FUNCTION_BLOCK AnlagenSequenz_06 (* Ring aus getrennter Vorlauf- und Nachlauf-Kette (je 5 Zwischenschritte) für 6 Motoren mit Störungs-Kaskade, s. KONZEPT_Anlagensequenz.md *)
  (* Standard: 61499-2; ApplicationDomain: Fördertechnik; Description: Copyright (c) 2026 HR Agrartechnik GmbH This program and the accompanying materials are made available under the terms of the Eclipse Public License 2.0 which is available at https://www.eclipse.org/legal/epl-2.0/ SPDX-License-Identifier: EPL-2.0 DRAFT (2026-08-12), 2. Fassung: Vorlauf und Nachlauf sind jetzt zwei getrennte, jeweils rein lineare Ketten (S_VOR1..S_VOR5 bzw. S_NACH1..S_NACH5), verbunden über S_AUS (unten) und S_LAEUFT (oben) zu einem Ring - anstelle der ersten Fassung mit 7 bidirektional genutzten Zuständen. Jeder Zustand hat dadurch genau einen festen Zeitwert (ZEk_EIN bzw. ZEk_AUS) und ein festes Motor-Muster, keine Richtungs-Fallunterscheidung mehr pro Zustand nötig. Bekannte, bewusste Vereinfachungen: 1) Jede STOERUNG_Mx hat ein eigenes Event EI_Mx (analog EO_Mx/DO_Mx), das direkt von jedem Zustand vor dem jeweiligen Zielschritt (S_NACH_x, bzw. S_AUS bei x=6) dorthin springt - kein Umweg mehr über einen Spiegelpunkt und kein Nachfassen über mehrere Zyklen. Ein AUS-Abbruch aus dem Vorlauf springt weiterhin auf den Spiegelpunkt (S_VOR_k -> S_NACH_(6-k)), da dort keine Motoren-Störung, sondern nur der Bedienerwunsch vorliegt. 2) Pro Motor gibt es ein Event EO_Mx mit angehängtem DO_Mx (analog EO_Sx/DO_Sx in sequence_T_04/_08). Der Baustein hat keine Selbstschleifen mehr (alle bisherigen liefen über das inzwischen entfernte EI_CYCLIC) - EO_Mx feuert also nur noch bei einem echten Zustandswechsel. 3) MaxBetriebRest/Nachlauf-Reste (Demo-Server-Schema) sind noch nicht abgebildet. *)
  (* Version 0.6, 2026-08-12, Franz Höpfinger, HR Agrartechnik GmbH *)
  PACKAGE logiBUS::utils::sequence::timed;
  IMPORT logiBUS::utils::sequence::const::sequence;
  IMPORT logiBUS::utils::sequence::const::sequence::NO_TIME;
  IMPORT logiBUS::utils::sequence::const::anlagenSequenz;
  IMPORT logiBUS::utils::sequence::const::anlagenSequenz::STATUS_BETRIEB_AUS;
  IMPORT logiBUS::utils::sequence::const::anlagenSequenz::STATUS_BETRIEB_HOCHFAHREN;
  IMPORT logiBUS::utils::sequence::const::anlagenSequenz::STATUS_BETRIEB_LAEUFT;
  IMPORT logiBUS::utils::sequence::const::anlagenSequenz::STATUS_BETRIEB_HERUNTERFAHREN;
  IMPORT logiBUS::utils::sequence::const::anlagenSequenz::STATUS_STOERUNG_KEINE;
  IMPORT logiBUS::utils::sequence::const::anlagenSequenz::STATUS_STOERUNG_AKTIV;
  IMPORT logiBUS::utils::sequence::const::anlagenSequenz::TRANSIT_ART_KEINE;
  IMPORT logiBUS::utils::sequence::const::anlagenSequenz::TRANSIT_ART_VORLAUF;
  IMPORT logiBUS::utils::sequence::const::anlagenSequenz::TRANSIT_ART_NACHLAUF;
  IMPORT logiBUS::utils::sequence::const::motorNummer;
  IMPORT logiBUS::utils::sequence::const::motorNummer::MOTOR_KEINER;
  IMPORT logiBUS::utils::sequence::const::motorNummer::MOTOR_M1;
  IMPORT logiBUS::utils::sequence::const::motorNummer::MOTOR_M2;
  IMPORT logiBUS::utils::sequence::const::motorNummer::MOTOR_M3;
  IMPORT logiBUS::utils::sequence::const::motorNummer::MOTOR_M4;
  IMPORT logiBUS::utils::sequence::const::motorNummer::MOTOR_M5;
  IMPORT logiBUS::utils::sequence::const::motorNummer::MOTOR_M6;
  IMPORT logiBUS::utils::sequence::const::zaehlstand;
  IMPORT logiBUS::utils::sequence::const::zaehlstand::ZAEHLSTAND_0;
  IMPORT logiBUS::utils::sequence::const::zaehlstand::ZAEHLSTAND_1;
  IMPORT logiBUS::utils::sequence::const::zaehlstand::ZAEHLSTAND_2;
  IMPORT logiBUS::utils::sequence::const::zaehlstand::ZAEHLSTAND_3;
  IMPORT logiBUS::utils::sequence::const::zaehlstand::ZAEHLSTAND_4;
  IMPORT logiBUS::utils::sequence::const::zaehlstand::ZAEHLSTAND_5;
  IMPORT logiBUS::utils::sequence::const::zaehlstand::ZAEHLSTAND_6;
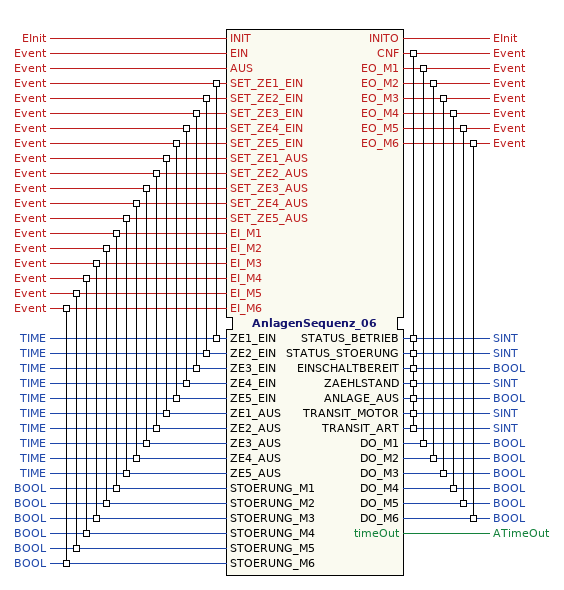
  EVENT_INPUT
    INIT : EInit; (* Initialization Request *)
    EIN; (* Startsequenz auslösen; nur wirksam wenn EINSCHALTBEREIT=TRUE; quittiert dabei zugleich eine anstehende Störungsanzeige *)
    AUS; (* Stopsequenz auslösen, aus jedem Schritt der Vorlauf-Kette oder aus S_LAEUFT *)
    SET_ZE1_EIN WITH ZE1_EIN; (* Update ZE1_EIN independently of EIN *)
    SET_ZE2_EIN WITH ZE2_EIN; (* Update ZE2_EIN independently of EIN *)
    SET_ZE3_EIN WITH ZE3_EIN; (* Update ZE3_EIN independently of EIN *)
    SET_ZE4_EIN WITH ZE4_EIN; (* Update ZE4_EIN independently of EIN *)
    SET_ZE5_EIN WITH ZE5_EIN; (* Update ZE5_EIN independently of EIN *)
    SET_ZE1_AUS WITH ZE1_AUS; (* Update ZE1_AUS independently of AUS *)
    SET_ZE2_AUS WITH ZE2_AUS; (* Update ZE2_AUS independently of AUS *)
    SET_ZE3_AUS WITH ZE3_AUS; (* Update ZE3_AUS independently of AUS *)
    SET_ZE4_AUS WITH ZE4_AUS; (* Update ZE4_AUS independently of AUS *)
    SET_ZE5_AUS WITH ZE5_AUS; (* Update ZE5_AUS independently of AUS *)
    EI_M1 WITH STOERUNG_M1; (* Störungsstatus Motor 1 hat sich geändert *)
    EI_M2 WITH STOERUNG_M2; (* Störungsstatus Motor 2 hat sich geändert *)
    EI_M3 WITH STOERUNG_M3; (* Störungsstatus Motor 3 hat sich geändert *)
    EI_M4 WITH STOERUNG_M4; (* Störungsstatus Motor 4 hat sich geändert *)
    EI_M5 WITH STOERUNG_M5; (* Störungsstatus Motor 5 hat sich geändert *)
    EI_M6 WITH STOERUNG_M6; (* Störungsstatus Motor 6 hat sich geändert *)
  END_EVENT
  EVENT_OUTPUT
    INITO : EInit; (* Initialization Confirm *)
    CNF WITH STATUS_BETRIEB, STATUS_STOERUNG, ZAEHLSTAND, EINSCHALTBEREIT, ANLAGE_AUS, TRANSIT_MOTOR, TRANSIT_ART; (* Ausführungsbestätigung, mit jedem Zustands-Update *)
    EO_M1 WITH DO_M1; (* Laufbefehl Motor 1 aktualisiert (analog EO_Sx in sequence_T_04/_08) *)
    EO_M2 WITH DO_M2; (* Laufbefehl Motor 2 aktualisiert *)
    EO_M3 WITH DO_M3; (* Laufbefehl Motor 3 aktualisiert *)
    EO_M4 WITH DO_M4; (* Laufbefehl Motor 4 aktualisiert *)
    EO_M5 WITH DO_M5; (* Laufbefehl Motor 5 aktualisiert *)
    EO_M6 WITH DO_M6; (* Laufbefehl Motor 6 aktualisiert *)
  END_EVENT
  VAR_INPUT
    ZE1_EIN : TIME := sequence::NO_TIME; (* S_VOR1 zu S_VOR2, M5 startet (Vorlauf) *)
    ZE2_EIN : TIME := sequence::NO_TIME; (* S_VOR2 zu S_VOR3, M4 startet (Vorlauf) *)
    ZE3_EIN : TIME := sequence::NO_TIME; (* S_VOR3 zu S_VOR4, M3 startet (Vorlauf) *)
    ZE4_EIN : TIME := sequence::NO_TIME; (* S_VOR4 zu S_VOR5, M2 startet (Vorlauf) *)
    ZE5_EIN : TIME := sequence::NO_TIME; (* S_VOR5 zu S_LAEUFT, M1 startet (Vorlauf) *)
    ZE1_AUS : TIME := sequence::NO_TIME; (* S_NACH1 zu S_NACH2, M2 stoppt (Nachlauf) *)
    ZE2_AUS : TIME := sequence::NO_TIME; (* S_NACH2 zu S_NACH3, M3 stoppt (Nachlauf) *)
    ZE3_AUS : TIME := sequence::NO_TIME; (* S_NACH3 zu S_NACH4, M4 stoppt (Nachlauf) *)
    ZE4_AUS : TIME := sequence::NO_TIME; (* S_NACH4 zu S_NACH5, M5 stoppt (Nachlauf) *)
    ZE5_AUS : TIME := sequence::NO_TIME; (* S_NACH5 zu S_AUS, M6 stoppt (Nachlauf) *)
    STOERUNG_M1 : BOOL := BOOL#FALSE; (* Motor 1 hat aktuell eine Störung anstehen *)
    STOERUNG_M2 : BOOL := BOOL#FALSE; (* Motor 2 hat aktuell eine Störung anstehen *)
    STOERUNG_M3 : BOOL := BOOL#FALSE; (* Motor 3 hat aktuell eine Störung anstehen *)
    STOERUNG_M4 : BOOL := BOOL#FALSE; (* Motor 4 hat aktuell eine Störung anstehen *)
    STOERUNG_M5 : BOOL := BOOL#FALSE; (* Motor 5 hat aktuell eine Störung anstehen *)
    STOERUNG_M6 : BOOL := BOOL#FALSE; (* Motor 6 hat aktuell eine Störung anstehen *)
  END_VAR
  VAR_OUTPUT
    STATUS_BETRIEB : SINT; (* 0=Aus 1=Hochfahren 2=Läuft 3=Herunterfahren *)
    STATUS_STOERUNG : SINT; (* 0=keine 4=aktiv, verriegelt bis EIN *)
    EINSCHALTBEREIT : BOOL; (* TRUE nur wenn alle Motoren stehen UND alle Motoren störungsfrei sind *)
    ZAEHLSTAND : SINT; (* 0..6, Anzahl aktuell laufender Motoren, s. Konzept *)
    ANLAGE_AUS : BOOL; (* TRUE nur in S_AUS (STATUS_BETRIEB = Aus) - Voraussetzung fuer Handbetrieb *)
    TRANSIT_MOTOR : SINT; (* 0 = keiner (S_AUS/S_LAEUFT), 1..6 = Motor-Nr., der nach Ablauf der aktuellen Zeit startet/stoppt (siehe TRANSIT_ART) *)
    TRANSIT_ART : SINT; (* anlagenSequenz::TRANSIT_ART_KEINE/_VORLAUF/_NACHLAUF *)
    DO_M1 : BOOL; (* Laufbefehl Motor 1 *)
    DO_M2 : BOOL; (* Laufbefehl Motor 2 *)
    DO_M3 : BOOL; (* Laufbefehl Motor 3 *)
    DO_M4 : BOOL; (* Laufbefehl Motor 4 *)
    DO_M5 : BOOL; (* Laufbefehl Motor 5 *)
    DO_M6 : BOOL; (* Laufbefehl Motor 6 *)
  END_VAR
  PLUGS
    timeOut : iec61499::events::ATimeOut; (* timeOut Adapter *)
  END_PLUGS
  EC_STATES
    xSTART; (* Initial State *)
    Init : -> INITO; (* Initialization *)
    sAUS : S_AUS_Setup, EI_CYCLIC_Auswertung, M1_AUS -> EO_M1, M2_AUS -> EO_M2, M3_AUS -> EO_M3, M4_AUS -> EO_M4, M5_AUS -> EO_M5, M6_AUS -> EO_M6, -> CNF; (* S_AUS, unten im Ring: keine Motoren laufen *)
    sVOR1 : S_VOR1_Setup, EI_CYCLIC_Auswertung, M1_AUS -> EO_M1, M2_AUS -> EO_M2, M3_AUS -> EO_M3, M4_AUS -> EO_M4, M5_AUS -> EO_M5, M6_EIN -> EO_M6, -> timeOut.START, -> CNF; (* S_VOR1 (Vorlauf-Kette): nur M6 läuft *)
    sVOR2 : S_VOR2_Setup, EI_CYCLIC_Auswertung, M1_AUS -> EO_M1, M2_AUS -> EO_M2, M3_AUS -> EO_M3, M4_AUS -> EO_M4, M5_EIN -> EO_M5, M6_EIN -> EO_M6, -> timeOut.START, -> CNF; (* S_VOR2 (Vorlauf-Kette): M5,M6 laufen *)
    sVOR3 : S_VOR3_Setup, EI_CYCLIC_Auswertung, M1_AUS -> EO_M1, M2_AUS -> EO_M2, M3_AUS -> EO_M3, M4_EIN -> EO_M4, M5_EIN -> EO_M5, M6_EIN -> EO_M6, -> timeOut.START, -> CNF; (* S_VOR3 (Vorlauf-Kette): M4,M5,M6 laufen *)
    sVOR4 : S_VOR4_Setup, EI_CYCLIC_Auswertung, M1_AUS -> EO_M1, M2_AUS -> EO_M2, M3_EIN -> EO_M3, M4_EIN -> EO_M4, M5_EIN -> EO_M5, M6_EIN -> EO_M6, -> timeOut.START, -> CNF; (* S_VOR4 (Vorlauf-Kette): M3,M4,M5,M6 laufen *)
    sVOR5 : S_VOR5_Setup, EI_CYCLIC_Auswertung, M1_AUS -> EO_M1, M2_EIN -> EO_M2, M3_EIN -> EO_M3, M4_EIN -> EO_M4, M5_EIN -> EO_M5, M6_EIN -> EO_M6, -> timeOut.START, -> CNF; (* S_VOR5 (Vorlauf-Kette): M2,M3,M4,M5,M6 laufen *)
    sLAEUFT : S_LAEUFT_Setup, EI_CYCLIC_Auswertung, M1_EIN -> EO_M1, M2_EIN -> EO_M2, M3_EIN -> EO_M3, M4_EIN -> EO_M4, M5_EIN -> EO_M5, M6_EIN -> EO_M6, -> CNF; (* S_LAEUFT, oben im Ring: alle 6 Motoren laufen *)
    sNACH1 : S_NACH1_Setup, EI_CYCLIC_Auswertung, M1_AUS -> EO_M1, M2_EIN -> EO_M2, M3_EIN -> EO_M3, M4_EIN -> EO_M4, M5_EIN -> EO_M5, M6_EIN -> EO_M6, -> timeOut.START, -> CNF; (* S_NACH1 (Nachlauf-Kette): M2,M3,M4,M5,M6 laufen (M1 gestoppt) *)
    sNACH2 : S_NACH2_Setup, EI_CYCLIC_Auswertung, M1_AUS -> EO_M1, M2_AUS -> EO_M2, M3_EIN -> EO_M3, M4_EIN -> EO_M4, M5_EIN -> EO_M5, M6_EIN -> EO_M6, -> timeOut.START, -> CNF; (* S_NACH2 (Nachlauf-Kette): M3,M4,M5,M6 laufen *)
    sNACH3 : S_NACH3_Setup, EI_CYCLIC_Auswertung, M1_AUS -> EO_M1, M2_AUS -> EO_M2, M3_AUS -> EO_M3, M4_EIN -> EO_M4, M5_EIN -> EO_M5, M6_EIN -> EO_M6, -> timeOut.START, -> CNF; (* S_NACH3 (Nachlauf-Kette): M4,M5,M6 laufen *)
    sNACH4 : S_NACH4_Setup, EI_CYCLIC_Auswertung, M1_AUS -> EO_M1, M2_AUS -> EO_M2, M3_AUS -> EO_M3, M4_AUS -> EO_M4, M5_EIN -> EO_M5, M6_EIN -> EO_M6, -> timeOut.START, -> CNF; (* S_NACH4 (Nachlauf-Kette): M5,M6 laufen *)
    sNACH5 : S_NACH5_Setup, EI_CYCLIC_Auswertung, M1_AUS -> EO_M1, M2_AUS -> EO_M2, M3_AUS -> EO_M3, M4_AUS -> EO_M4, M5_AUS -> EO_M5, M6_EIN -> EO_M6, -> timeOut.START, -> CNF; (* S_NACH5 (Nachlauf-Kette): nur M6 läuft *)
  END_STATES
  EC_TRANSITIONS
    sAUS TO sVOR1 := EIN[NOT (STOERUNG_M1 OR STOERUNG_M2 OR STOERUNG_M3 OR STOERUNG_M4 OR STOERUNG_M5 OR STOERUNG_M6)];
    sVOR1 TO sVOR2 := timeOut.TimeOut;
    sVOR1 TO sNACH5 := AUS;
    sVOR1 TO sNACH1 := EI_M1[STOERUNG_M1];
    sVOR1 TO sNACH2 := EI_M2[STOERUNG_M2];
    sVOR1 TO sNACH3 := EI_M3[STOERUNG_M3];
    sVOR1 TO sNACH4 := EI_M4[STOERUNG_M4];
    sVOR1 TO sNACH5 := EI_M5[STOERUNG_M5];
    sVOR1 TO sAUS := EI_M6[STOERUNG_M6];
    sVOR2 TO sVOR3 := timeOut.TimeOut;
    sVOR2 TO sNACH4 := AUS;
    sVOR2 TO sNACH1 := EI_M1[STOERUNG_M1];
    sVOR2 TO sNACH2 := EI_M2[STOERUNG_M2];
    sVOR2 TO sNACH3 := EI_M3[STOERUNG_M3];
    sVOR2 TO sNACH4 := EI_M4[STOERUNG_M4];
    sVOR2 TO sNACH5 := EI_M5[STOERUNG_M5];
    sVOR2 TO sAUS := EI_M6[STOERUNG_M6];
    sVOR3 TO sVOR4 := timeOut.TimeOut;
    sVOR3 TO sNACH3 := AUS;
    sVOR3 TO sNACH1 := EI_M1[STOERUNG_M1];
    sVOR3 TO sNACH2 := EI_M2[STOERUNG_M2];
    sVOR3 TO sNACH3 := EI_M3[STOERUNG_M3];
    sVOR3 TO sNACH4 := EI_M4[STOERUNG_M4];
    sVOR3 TO sNACH5 := EI_M5[STOERUNG_M5];
    sVOR3 TO sAUS := EI_M6[STOERUNG_M6];
    sVOR4 TO sVOR5 := timeOut.TimeOut;
    sVOR4 TO sNACH2 := AUS;
    sVOR4 TO sNACH1 := EI_M1[STOERUNG_M1];
    sVOR4 TO sNACH2 := EI_M2[STOERUNG_M2];
    sVOR4 TO sNACH3 := EI_M3[STOERUNG_M3];
    sVOR4 TO sNACH4 := EI_M4[STOERUNG_M4];
    sVOR4 TO sNACH5 := EI_M5[STOERUNG_M5];
    sVOR4 TO sAUS := EI_M6[STOERUNG_M6];
    sVOR5 TO sLAEUFT := timeOut.TimeOut;
    sVOR5 TO sNACH1 := AUS;
    sVOR5 TO sNACH1 := EI_M1[STOERUNG_M1];
    sVOR5 TO sNACH2 := EI_M2[STOERUNG_M2];
    sVOR5 TO sNACH3 := EI_M3[STOERUNG_M3];
    sVOR5 TO sNACH4 := EI_M4[STOERUNG_M4];
    sVOR5 TO sNACH5 := EI_M5[STOERUNG_M5];
    sVOR5 TO sAUS := EI_M6[STOERUNG_M6];
    sLAEUFT TO sNACH1 := AUS;
    sLAEUFT TO sNACH1 := EI_M1[STOERUNG_M1];
    sLAEUFT TO sNACH2 := EI_M2[STOERUNG_M2];
    sLAEUFT TO sNACH3 := EI_M3[STOERUNG_M3];
    sLAEUFT TO sNACH4 := EI_M4[STOERUNG_M4];
    sLAEUFT TO sNACH5 := EI_M5[STOERUNG_M5];
    sLAEUFT TO sAUS := EI_M6[STOERUNG_M6];
    sNACH1 TO sNACH2 := timeOut.TimeOut;
    sNACH1 TO sNACH2 := EI_M2[STOERUNG_M2];
    sNACH1 TO sNACH3 := EI_M3[STOERUNG_M3];
    sNACH1 TO sNACH4 := EI_M4[STOERUNG_M4];
    sNACH1 TO sNACH5 := EI_M5[STOERUNG_M5];
    sNACH1 TO sAUS := EI_M6[STOERUNG_M6];
    sNACH2 TO sNACH3 := timeOut.TimeOut;
    sNACH2 TO sNACH3 := EI_M3[STOERUNG_M3];
    sNACH2 TO sNACH4 := EI_M4[STOERUNG_M4];
    sNACH2 TO sNACH5 := EI_M5[STOERUNG_M5];
    sNACH2 TO sAUS := EI_M6[STOERUNG_M6];
    sNACH3 TO sNACH4 := timeOut.TimeOut;
    sNACH3 TO sNACH4 := EI_M4[STOERUNG_M4];
    sNACH3 TO sNACH5 := EI_M5[STOERUNG_M5];
    sNACH3 TO sAUS := EI_M6[STOERUNG_M6];
    sNACH4 TO sNACH5 := timeOut.TimeOut;
    sNACH4 TO sNACH5 := EI_M5[STOERUNG_M5];
    sNACH4 TO sAUS := EI_M6[STOERUNG_M6];
    sNACH5 TO sAUS := timeOut.TimeOut;
    sNACH5 TO sAUS := EI_M6[STOERUNG_M6];
    sVOR1 TO sVOR1 := SET_ZE1_EIN;
    sVOR2 TO sVOR2 := SET_ZE2_EIN;
    sVOR3 TO sVOR3 := SET_ZE3_EIN;
    sVOR4 TO sVOR4 := SET_ZE4_EIN;
    sVOR5 TO sVOR5 := SET_ZE5_EIN;
    sNACH1 TO sNACH1 := SET_ZE1_AUS;
    sNACH2 TO sNACH2 := SET_ZE2_AUS;
    sNACH3 TO sNACH3 := SET_ZE3_AUS;
    sNACH4 TO sNACH4 := SET_ZE4_AUS;
    sNACH5 TO sNACH5 := SET_ZE5_AUS;
    xSTART TO Init := INIT;
    Init TO sAUS := 1;
  END_TRANSITIONS
  ALGORITHM initialize IN ST: (* Initialization algorithm *)

  END_ALGORITHM
  ALGORITHM deInitialize IN ST: (* Normally executed algorithm *)

  END_ALGORITHM
  ALGORITHM EI_CYCLIC_Auswertung IN ST: (* Liest STOERUNG_M1..M6 neu ein, setzt STATUS_STOERUNG falls eine aktiv ist, und berechnet EINSCHALTBEREIT/ANLAGE_AUS *)
// Störungssignale frisch einlesen (BOOL-Dauersignale, kein Event-Consumption-Problem, s. Konzept
// Frage 4)
IF STOERUNG_M1 OR STOERUNG_M2 OR STOERUNG_M3 OR STOERUNG_M4 OR STOERUNG_M5 OR STOERUNG_M6 THEN
	STATUS_STOERUNG := anlagenSequenz::STATUS_STOERUNG_AKTIV; // verriegelt bis zur nächsten erfolgreichen EIN-Quittierung
END_IF;

// Einschaltbereit: alle Motoren stehen (S_AUS) UND alle Motoren aktuell (live) störungsfrei.
// Bewusst NICHT an STATUS_STOERUNG gekoppelt: das bleibt bis zum naechsten EIN verriegelt, EIN
// selbst kommt aber nur an, wenn EINSCHALTBEREIT die Visu-Sperre freigibt - sonst Deadlock.
EINSCHALTBEREIT := (ZAEHLSTAND = 0)
	AND NOT (STOERUNG_M1 OR STOERUNG_M2 OR STOERUNG_M3 OR STOERUNG_M4 OR STOERUNG_M5 OR STOERUNG_M6);

// Voraussetzung fuer Handbetrieb: nur wenn die Anlage wirklich in S_AUS steht (unabhaengig von
// Stoerungen - eine Stoerung soll Handbetrieb zum Freifahren nicht zusaetzlich blockieren).
ANLAGE_AUS := (STATUS_BETRIEB = anlagenSequenz::STATUS_BETRIEB_AUS);
  END_ALGORITHM
  ALGORITHM M1_EIN IN ST: (* Setzt den Laufbefehl DO_M1 auf TRUE (Motor 1 einschalten) *)
DO_M1 := BOOL#TRUE;
  END_ALGORITHM
  ALGORITHM M1_AUS IN ST: (* Setzt den Laufbefehl DO_M1 auf FALSE (Motor 1 ausschalten) *)
DO_M1 := BOOL#FALSE;
  END_ALGORITHM
  ALGORITHM M2_EIN IN ST: (* Setzt den Laufbefehl DO_M2 auf TRUE (Motor 2 einschalten) *)
DO_M2 := BOOL#TRUE;
  END_ALGORITHM
  ALGORITHM M2_AUS IN ST: (* Setzt den Laufbefehl DO_M2 auf FALSE (Motor 2 ausschalten) *)
DO_M2 := BOOL#FALSE;
  END_ALGORITHM
  ALGORITHM M3_EIN IN ST: (* Setzt den Laufbefehl DO_M3 auf TRUE (Motor 3 einschalten) *)
DO_M3 := BOOL#TRUE;
  END_ALGORITHM
  ALGORITHM M3_AUS IN ST: (* Setzt den Laufbefehl DO_M3 auf FALSE (Motor 3 ausschalten) *)
DO_M3 := BOOL#FALSE;
  END_ALGORITHM
  ALGORITHM M4_EIN IN ST: (* Setzt den Laufbefehl DO_M4 auf TRUE (Motor 4 einschalten) *)
DO_M4 := BOOL#TRUE;
  END_ALGORITHM
  ALGORITHM M4_AUS IN ST: (* Setzt den Laufbefehl DO_M4 auf FALSE (Motor 4 ausschalten) *)
DO_M4 := BOOL#FALSE;
  END_ALGORITHM
  ALGORITHM M5_EIN IN ST: (* Setzt den Laufbefehl DO_M5 auf TRUE (Motor 5 einschalten) *)
DO_M5 := BOOL#TRUE;
  END_ALGORITHM
  ALGORITHM M5_AUS IN ST: (* Setzt den Laufbefehl DO_M5 auf FALSE (Motor 5 ausschalten) *)
DO_M5 := BOOL#FALSE;
  END_ALGORITHM
  ALGORITHM M6_EIN IN ST: (* Setzt den Laufbefehl DO_M6 auf TRUE (Motor 6 einschalten) *)
DO_M6 := BOOL#TRUE;
  END_ALGORITHM
  ALGORITHM M6_AUS IN ST: (* Setzt den Laufbefehl DO_M6 auf FALSE (Motor 6 ausschalten) *)
DO_M6 := BOOL#FALSE;
  END_ALGORITHM
  ALGORITHM S_AUS_Setup IN ST: (* Setup für S_AUS: ZAEHLSTAND auf 0, STATUS_BETRIEB auf Aus - keine Motoren laufen, Ring-Grundzustand *)
// S_AUS: keine Motoren laufen
ZAEHLSTAND := zaehlstand::ZAEHLSTAND_0;
STATUS_BETRIEB := anlagenSequenz::STATUS_BETRIEB_AUS;
TRANSIT_MOTOR := motorNummer::MOTOR_KEINER;
TRANSIT_ART := anlagenSequenz::TRANSIT_ART_KEINE;
  END_ALGORITHM
  ALGORITHM S_VOR1_Setup IN ST: (* Setup für S_VOR1: ZAEHLSTAND auf 1, STATUS_BETRIEB auf Hochfahren, quittiert STATUS_STOERUNG (nur über EIN erreichbar) und lädt Timer ZE1_EIN für den nächsten Vorlauf-Schritt *)
// S_VOR1: M6 läuft
ZAEHLSTAND := zaehlstand::ZAEHLSTAND_1;
STATUS_BETRIEB := anlagenSequenz::STATUS_BETRIEB_HOCHFAHREN;
STATUS_STOERUNG := anlagenSequenz::STATUS_STOERUNG_KEINE; // Quittierung: EIN wurde soeben angenommen (S_VOR1 ist nur über EIN erreichbar)
timeOut.DT := ZE1_EIN;
TRANSIT_MOTOR := motorNummer::MOTOR_M5;
TRANSIT_ART := anlagenSequenz::TRANSIT_ART_VORLAUF;
  END_ALGORITHM
  ALGORITHM S_VOR2_Setup IN ST: (* Setup für S_VOR2: ZAEHLSTAND auf 2, STATUS_BETRIEB auf Hochfahren, lädt Timer ZE2_EIN für den nächsten Vorlauf-Schritt *)
// S_VOR2: M5,M6 laufen
ZAEHLSTAND := zaehlstand::ZAEHLSTAND_2;
STATUS_BETRIEB := anlagenSequenz::STATUS_BETRIEB_HOCHFAHREN;
timeOut.DT := ZE2_EIN;
TRANSIT_MOTOR := motorNummer::MOTOR_M4;
TRANSIT_ART := anlagenSequenz::TRANSIT_ART_VORLAUF;
  END_ALGORITHM
  ALGORITHM S_VOR3_Setup IN ST: (* Setup für S_VOR3: ZAEHLSTAND auf 3, STATUS_BETRIEB auf Hochfahren, lädt Timer ZE3_EIN für den nächsten Vorlauf-Schritt *)
// S_VOR3: M4,M5,M6 laufen
ZAEHLSTAND := zaehlstand::ZAEHLSTAND_3;
STATUS_BETRIEB := anlagenSequenz::STATUS_BETRIEB_HOCHFAHREN;
timeOut.DT := ZE3_EIN;
TRANSIT_MOTOR := motorNummer::MOTOR_M3;
TRANSIT_ART := anlagenSequenz::TRANSIT_ART_VORLAUF;
  END_ALGORITHM
  ALGORITHM S_VOR4_Setup IN ST: (* Setup für S_VOR4: ZAEHLSTAND auf 4, STATUS_BETRIEB auf Hochfahren, lädt Timer ZE4_EIN für den nächsten Vorlauf-Schritt *)
// S_VOR4: M3,M4,M5,M6 laufen
ZAEHLSTAND := zaehlstand::ZAEHLSTAND_4;
STATUS_BETRIEB := anlagenSequenz::STATUS_BETRIEB_HOCHFAHREN;
timeOut.DT := ZE4_EIN;
TRANSIT_MOTOR := motorNummer::MOTOR_M2;
TRANSIT_ART := anlagenSequenz::TRANSIT_ART_VORLAUF;
  END_ALGORITHM
  ALGORITHM S_VOR5_Setup IN ST: (* Setup für S_VOR5: ZAEHLSTAND auf 5, STATUS_BETRIEB auf Hochfahren, lädt Timer ZE5_EIN für den letzten Vorlauf-Schritt (M1 startet danach) *)
// S_VOR5: M2,M3,M4,M5,M6 laufen
ZAEHLSTAND := zaehlstand::ZAEHLSTAND_5;
STATUS_BETRIEB := anlagenSequenz::STATUS_BETRIEB_HOCHFAHREN;
timeOut.DT := ZE5_EIN;
TRANSIT_MOTOR := motorNummer::MOTOR_M1;
TRANSIT_ART := anlagenSequenz::TRANSIT_ART_VORLAUF;
  END_ALGORITHM
  ALGORITHM S_LAEUFT_Setup IN ST: (* Setup für S_LAEUFT: ZAEHLSTAND auf 6, STATUS_BETRIEB auf Läuft - alle 6 Motoren laufen, oberer Ring-Zustand *)
// S_LAEUFT: alle 6 Motoren laufen
ZAEHLSTAND := zaehlstand::ZAEHLSTAND_6;
STATUS_BETRIEB := anlagenSequenz::STATUS_BETRIEB_LAEUFT;
TRANSIT_MOTOR := motorNummer::MOTOR_KEINER;
TRANSIT_ART := anlagenSequenz::TRANSIT_ART_KEINE;
  END_ALGORITHM
  ALGORITHM S_NACH1_Setup IN ST: (* Setup für S_NACH1: ZAEHLSTAND auf 5, STATUS_BETRIEB auf Herunterfahren, lädt den Nachlauf-Timer ZE1_AUS *)
// S_NACH1: M2,M3,M4,M5,M6 laufen (M1 gestoppt)
ZAEHLSTAND := zaehlstand::ZAEHLSTAND_5;
STATUS_BETRIEB := anlagenSequenz::STATUS_BETRIEB_HERUNTERFAHREN;
timeOut.DT := ZE1_AUS;
TRANSIT_MOTOR := motorNummer::MOTOR_M2;
TRANSIT_ART := anlagenSequenz::TRANSIT_ART_NACHLAUF;
  END_ALGORITHM
  ALGORITHM S_NACH2_Setup IN ST: (* Setup für S_NACH2: ZAEHLSTAND auf 4, STATUS_BETRIEB auf Herunterfahren, lädt den Nachlauf-Timer ZE2_AUS *)
// S_NACH2: M3,M4,M5,M6 laufen
ZAEHLSTAND := zaehlstand::ZAEHLSTAND_4;
STATUS_BETRIEB := anlagenSequenz::STATUS_BETRIEB_HERUNTERFAHREN;
timeOut.DT := ZE2_AUS;
TRANSIT_MOTOR := motorNummer::MOTOR_M3;
TRANSIT_ART := anlagenSequenz::TRANSIT_ART_NACHLAUF;
  END_ALGORITHM
  ALGORITHM S_NACH3_Setup IN ST: (* Setup für S_NACH3: ZAEHLSTAND auf 3, STATUS_BETRIEB auf Herunterfahren, lädt den Nachlauf-Timer ZE3_AUS *)
// S_NACH3: M4,M5,M6 laufen
ZAEHLSTAND := zaehlstand::ZAEHLSTAND_3;
STATUS_BETRIEB := anlagenSequenz::STATUS_BETRIEB_HERUNTERFAHREN;
timeOut.DT := ZE3_AUS;
TRANSIT_MOTOR := motorNummer::MOTOR_M4;
TRANSIT_ART := anlagenSequenz::TRANSIT_ART_NACHLAUF;
  END_ALGORITHM
  ALGORITHM S_NACH4_Setup IN ST: (* Setup für S_NACH4: ZAEHLSTAND auf 2, STATUS_BETRIEB auf Herunterfahren, lädt den Nachlauf-Timer ZE4_AUS *)
// S_NACH4: M5,M6 laufen
ZAEHLSTAND := zaehlstand::ZAEHLSTAND_2;
STATUS_BETRIEB := anlagenSequenz::STATUS_BETRIEB_HERUNTERFAHREN;
timeOut.DT := ZE4_AUS;
TRANSIT_MOTOR := motorNummer::MOTOR_M5;
TRANSIT_ART := anlagenSequenz::TRANSIT_ART_NACHLAUF;
  END_ALGORITHM
  ALGORITHM S_NACH5_Setup IN ST: (* Setup für S_NACH5: ZAEHLSTAND auf 1, STATUS_BETRIEB auf Herunterfahren, lädt den Nachlauf-Timer ZE5_AUS (letzter Schritt vor S_AUS) *)
// S_NACH5: nur M6 läuft
ZAEHLSTAND := zaehlstand::ZAEHLSTAND_1;
STATUS_BETRIEB := anlagenSequenz::STATUS_BETRIEB_HERUNTERFAHREN;
timeOut.DT := ZE5_AUS;
TRANSIT_MOTOR := motorNummer::MOTOR_M6;
TRANSIT_ART := anlagenSequenz::TRANSIT_ART_NACHLAUF;
  END_ALGORITHM
END_FUNCTION_BLOCK
